FUNCTION_BLOCK POU_2
VAR_INPUT
END_VAR
VAR_OUTPUT
END_VAR
VAR
END_VAR

END_FUNCTION_BLOCK

(* stored: Version 1.1.0.1, ProductVersion 3.1.4024.13
   POU POU_2: Id {3eb8aa00-9a33-483d-b7d8-e09c1dffc10f}, SpecialFunc None *)
